{attribute 'GeneratedUsingTerminal: EL1262-0000-0002'}
{attribute addProperty BoxType "EL1262-0000-0002"}
{attribute addProperty Id "StartTimeNextLatchAT %I*UDINT4"}
{attribute addProperty CRC "3994574359"}
{attribute addProperty Size "4"}
TYPE NextSync1Time_EE185E17 EXTENDS InputBase_8311D824 :
STRUCT
	{attribute addProperty Name "StartTimeNextLatch"}
	StartTimeNextLatch AT %I* : UDINT;
END_STRUCT
END_TYPE

(* stored: Version 1.2.0.0, ProductVersion 3.1.4024.11
   DUT NextSync1Time_EE185E17: Id {da80e48f-43a8-4235-90f2-f7fbb20cc22e} *)
